TYPE ST_UN_CleanroomConnectSettings :
STRUCT
	stPalletConveyor : ST_SettingsPalletConveyor;
	stDockingInterface : ST_SettingsDockingInterface;
	stLiftingTransport : ST_SettingsLiftingTransport;
	stAirTreatment : ST_SettingsAirTreatment;
END_STRUCT
END_TYPE

(* stored: Version 1.1.0.1, ProductVersion 3.1.4024.12
   DUT ST_UN_CleanroomConnectSettings: Id {3f2f6cc8-3931-41b6-b35a-8f99944d8bca} *)
